Staubli VAL3: PickAndPlace.pgx

program PickAndPlace()
      while true
        movej(pp1, flange, mNomSpeed)
        movej(pp2, flange, mNomSpeed)
        movej(pp3, flange, mNomSpeed)
        movej(pp4, flange, mNomSpeed)
        waitEndMove()
      endWhile
